{attribute addProperty BoxType "EK1122-0000-0018"}
{attribute addProperty Id "Beckhoff_APS4xxxsub_EK1100EK1100_179A0949162A_0001_APS4322_7000_0017APS4322_C8B6F1122256282"}
{attribute addProperty CRC "2839132900"}
{attribute addProperty SizeInBites "2272"}
{attribute addProperty SizeInBytes "284"}
TYPE Beckhoff_APS4xxxEK1122_A939BAE4 EXTENDS EK1122_179A0949 :
STRUCT
	{attribute addProperty Name "Beckhoff_APS4xxxsub_EK1100"}
	Beckhoff_APS4xxxsub_EK1100 : EK1100_179A0949;
	{attribute addProperty Name "A_0001_APS4322_7000_0017"}
	A_0001_APS4322_7000_0017 : APS4322_C8B6F112;
END_STRUCT
END_TYPE

(* stored: Version 1.2.0.0, ProductVersion 3.1.4024.9
   DUT Beckhoff_APS4xxxEK1122_A939BAE4: Id {37575bc9-87e3-40a9-be21-32f0f60f5962} *)
